// TIA Portal V17 export
// export: Created 2025-06-26T07:49:40.3880186Z, ExportSetting WithDefaults, DisplayName Totally Integrated Automation Portal, DisplayVersion V17 Update 8, DisplayName TIA Portal Openness, DisplayVersion V17 Update 8, DisplayName TIA Portal Version Control Interface, DisplayVersion V17, DisplayName STEP 7 Professional, DisplayVersion V17 Update 8, DisplayName STEP 7 Safety, DisplayVersion V17 Update 6, DisplayName WinCC Advanced, DisplayVersion V17 Update 8
FUNCTION_BLOCK "OperatingTimeCounters"   // FB41, FBD
{ S7_Optimized_Access := 'TRUE' }
VERSION : 0.1
// stored: AutoNumber true, IsIECCheckEnabled false, IsRetainMemResEnabled false, MemoryReserve 0, SetENOAutomatically false, UDAEnableTagReadback false
   VAR
      SystemOnTime { ExternalAccessible := 'False'; ExternalVisible := 'False'; ExternalWritable := 'False'} : "fbHoursCounter";
      SwitchedOnTime { ExternalAccessible := 'False'; ExternalVisible := 'False'; ExternalWritable := 'False'; S7_SetPoint := 'True'} : "fbHoursCounter";
      RunningTime { ExternalAccessible := 'False'; ExternalVisible := 'False'; ExternalWritable := 'False'; S7_SetPoint := 'True'} : "fbHoursCounter";
      RuntimeMemory { ExternalAccessible := 'False'; ExternalVisible := 'False'; ExternalWritable := 'False'; S7_SetPoint := 'True'} : LReal;
   END_VAR
BEGIN

REGION Network 1: Read out scan time
   // This is in the wrong place
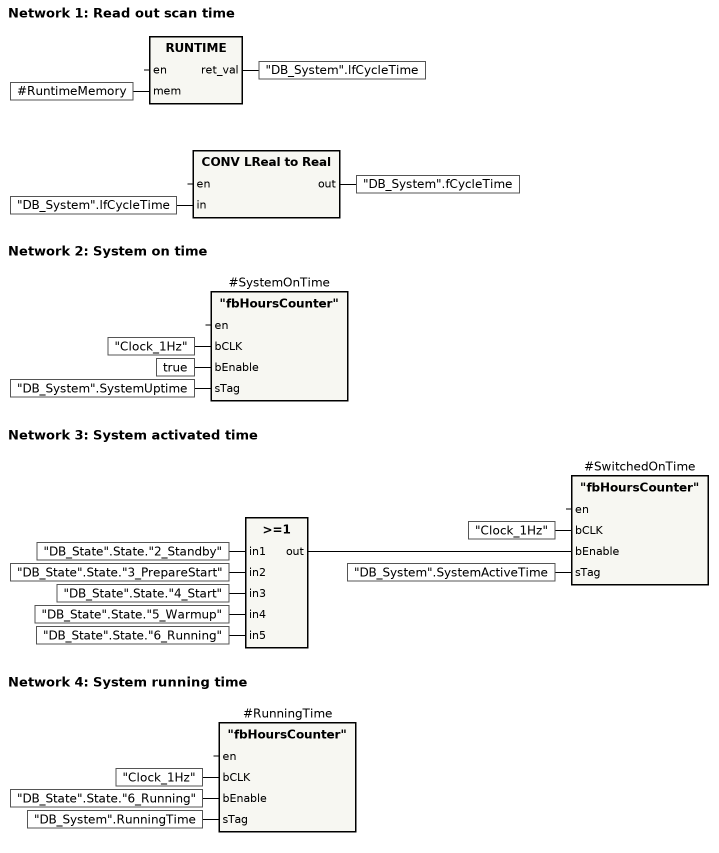
   // no SCL statement known for Runtime: written as a call
   "DB_System".lfCycleTime := Runtime(mem := #RuntimeMemory);
   "DB_System".fCycleTime := LREAL_TO_REAL("DB_System".lfCycleTime);
END_REGION

REGION Network 2: System on time
   #SystemOnTime(bCLK := "Clock_1Hz", bEnable := true, sTag := "DB_System".SystemUptime);   // "fbHoursCounter"
END_REGION

REGION Network 3: System activated time
   #SwitchedOnTime(bCLK := "Clock_1Hz",   // "fbHoursCounter"
                   bEnable := "DB_State".State."2_Standby" OR "DB_State".State."3_PrepareStart" OR "DB_State".State."4_Start" OR "DB_State".State."5_Warmup" OR "DB_State".State."6_Running",
                   sTag := "DB_System".SystemActiveTime);
END_REGION

REGION Network 4: System running time
   #RunningTime(bCLK := "Clock_1Hz", bEnable := "DB_State".State."6_Running", sTag := "DB_System".RunningTime);   // "fbHoursCounter"
END_REGION
END_FUNCTION_BLOCK
